FUNCTION_BLOCK FB_MoveRequest_TestDouble IMPLEMENTS I_MoveRequest
VAR
    eEnableMode: E_StageEnableMode:=E_StageEnableMode.DURING_MOTION;
    bMoveCmd	: BOOL;
    bHomeCmd: BOOL;
    eHomeMode	: E_EpicsHomeCmd;
    bEnableDone : BOOL;
    bMoveOk: BOOL;
    bExecute : BOOL;
    stMotionRequestStatus : ST_MoveRequestStatus;
END_VAR

{warning 'Add method implementation '}
METHOD ClearMoveRequest
END_METHOD

{warning 'Add method implementation '}
METHOD ClearMoveRequestErrors
END_METHOD

{warning 'Add property implementation'}
PROPERTY EnableMode : ENUM_StageEnableMode
GET
END_GET
SET
END_SET
END_PROPERTY

PROPERTY INTERNAL EpicsMotorCommand : INT
GET
EpicsMotorCommand := stMotionRequestStatus.nCommand;
END_GET
SET
stMotionRequestStatus.nCommand := EpicsMotorCommand;
END_SET
END_PROPERTY

{warning 'Add method implementation '}
METHOD HaltMoveRequest : BOOL
VAR_INPUT
    Busy	: BOOL;
END_VAR
END_METHOD

{warning 'Add method implementation '}
METHOD InitMoveRequest
END_METHOD

{warning 'Add method implementation '}
METHOD MoveRequest
VAR_INPUT
    (* From Axis through the drive*)
    EnableDone	: BOOL;
    (* From Interlock through the drive*)
    MoveOk	: BOOL;
END_VAR
END_METHOD

{warning 'Add method implementation '}
METHOD MoveRequestCompleted
VAR_INPUT
    MoveDone	: BOOL;
    HomeDone	: BOOL;
END_VAR
END_METHOD

{warning 'Add method implementation '}
METHOD MoveRequestDone
VAR_INPUT
    Done	: BOOL;
END_VAR
END_METHOD

{warning 'Add method implementation '}
METHOD MoveRequestError
VAR_INPUT
    Error	: BOOL;
    ErrorId	: UDINT;
    ErrorMessage	: T_MAXSTRING;
END_VAR
END_METHOD

{warning 'Add method implementation '}
METHOD MoveResetDone
END_METHOD

{warning 'Add method implementation '}
METHOD ResetMoveEnable
END_METHOD

{warning 'Add method implementation '}
METHOD ResetMoveRequest
END_METHOD

METHOD RestoreSettings
VAR_INPUT
    RestoreDone : BOOL;
    SavedPosition : LREAL;
END_VAR
END_METHOD

{warning 'Add property implementation'}
PROPERTY Status : REFERENCE TO ST_MoveRequestStatus
GET
Status REF= stMotionRequestStatus;
END_GET
END_PROPERTY

END_FUNCTION_BLOCK

(* stored: Version 1.1.0.1
   POU FB_MoveRequest_TestDouble: Id {f79ff9ea-c5fb-4287-a47e-3e52fe39dad4}, SpecialFunc None
   Method ClearMoveRequest: Id {8bff28f3-fae6-46e5-8f37-8cf755f60759}
   Method ClearMoveRequestErrors: Id {a7158e7f-c22a-418f-a7c6-dc5045d8a707}
   Property EnableMode: Id {66b8f19e-4221-443f-b49c-d49ffdab97f1}
   Get Get: Id {a1b2d88c-6b31-492d-ab0b-905dfac6e434}
   Set Set: Id {0826e199-470b-41c3-a9c0-813d50acad62}
   Property EpicsMotorCommand: Id {9e3a0522-4957-4a0f-822b-ec71ef18e062}
   Get Get: Id {3e155d13-93f5-474c-9ebd-b644c33d821d}
   Set Set: Id {ad667525-86b7-4afb-af24-f093ed7473d3}
   Method HaltMoveRequest: Id {62f53f48-84cf-46cf-967e-c760a56f5485}
   Method InitMoveRequest: Id {26231f67-3b3b-4070-a264-798d1d19bc23}
   Method MoveRequest: Id {e51e3678-c3aa-4bd6-8679-36a860fb753b}
   Method MoveRequestCompleted: Id {c7ab1522-b76e-48c4-86bd-f5dd13d1298b}
   Method MoveRequestDone: Id {44c9f40d-ce58-4660-9fa7-f17f0c4adf10}
   Method MoveRequestError: Id {17958167-de04-4369-8ecb-b80a6455af92}
   Method MoveResetDone: Id {898f0db3-7029-4aa3-bbce-939166937d7c}
   Method ResetMoveEnable: Id {d9a38b2c-4208-4dbc-9ad7-b8bdcfa1e4f3}
   Method ResetMoveRequest: Id {d9033c6c-929e-4449-ae64-e4cd6df1d3c0}
   Method RestoreSettings: Id {41457382-4ca7-41b9-9de4-5889425b6779}
   Property Status: Id {aa3ec75e-548d-4120-aabb-5680dda6acfd}
   Get Get: Id {e6adfc98-9c8d-4e29-8b25-b75a7be4044a} *)
